# EPICS substitutions: ek9000App/Db/EL4102.substitutions
file EL4102.template
{       pattern
        {
                TERMINAL,

        }
        {
        }
}
